PROGRAM B_Program
VAR
	x : LREAL;
	x_inc : LREAL := 0.0001;
END_VAR

x := x + x_inc;

END_PROGRAM

(* stored: Version 1.1.0.1, ProductVersion 3.1.4025.12
   POU B_Program: Id {4d82e6e2-c3b8-45cf-af6c-b81d6b859706}, SpecialFunc None *)
